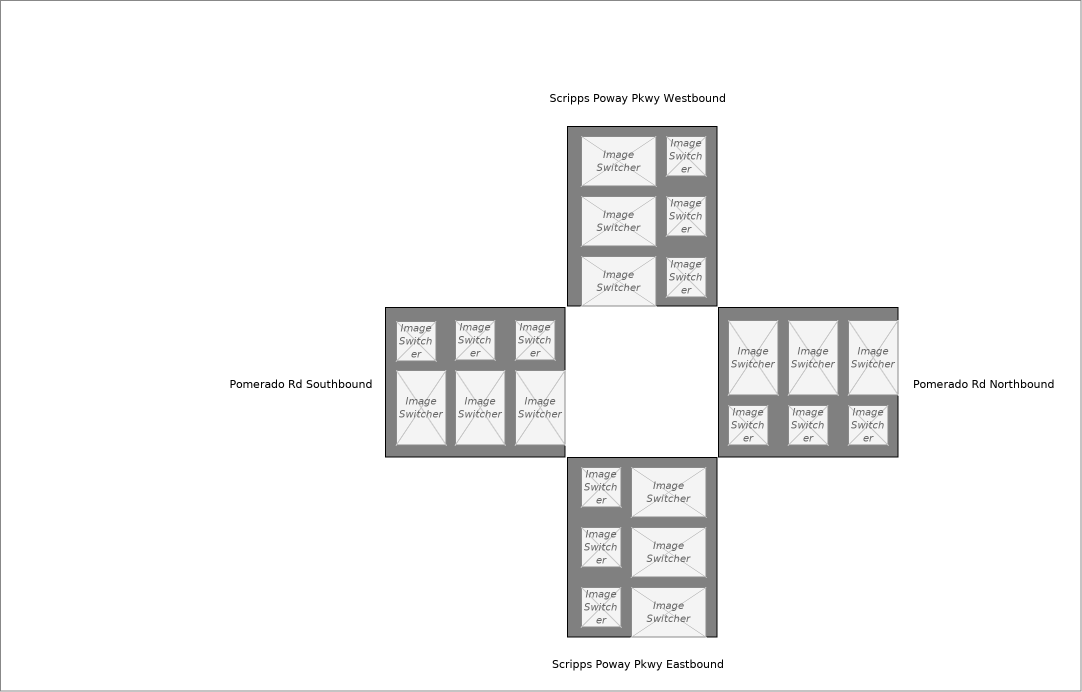
VISUALIZATION Initial_Intersection_Visualization  // 1082x692
    Group (203,71 879x566)
        Group (182,55 513x511)
            Group (182,331 150x180)
                RoundedRectangle (0,0 150x180)
                ImageSwitcher (64,70 75x50), variable: MAIN.fb_Major_Street_Forward_Phase_6.b_Yellow_Signal_Active, behaviour: TOGGLE
                ImageSwitcher (64,130 75x50), variable: MAIN.fb_Major_Street_Forward_Phase_6.b_Green_Signal_Active, behaviour: TOGGLE
                ImageSwitcher (64,10 75x50), variable: MAIN.fb_Major_Street_Forward_Phase_6.b_Red_Signal_Active, behaviour: TOGGLE
                ImageSwitcher (14,10 40x40), variable: MAIN.fb_Major_Street_Left_Turn_Phase_1.b_Red_Signal_Active, behaviour: TOGGLE
                ImageSwitcher (14,70 40x40), variable: MAIN.fb_Major_Street_Left_Turn_Phase_1.b_Yellow_Signal_Active, behaviour: TOGGLE
                ImageSwitcher (14,130 40x40), variable: MAIN.fb_Major_Street_Left_Turn_Phase_1.b_Green_Signal_Active, behaviour: TOGGLE
            Group (333,181 180x150)
                RoundedRectangle (0,0 180x150)
                Group (10,13 170x125)
                    ImageSwitcher (0,0 50x75), variable: MAIN.fb_Minor_Street_Forward_Phase_4.b_Red_Signal_Active, behaviour: TOGGLE
                    ImageSwitcher (60,0 50x75), variable: MAIN.fb_Minor_Street_Forward_Phase_4.b_Yellow_Signal_Active, behaviour: TOGGLE
                    ImageSwitcher (120,0 50x75), variable: MAIN.fb_Minor_Street_Forward_Phase_4.b_Green_Signal_Active, behaviour: TOGGLE
                    ImageSwitcher (0,85 40x40), variable: MAIN.fb_Minor_Street_Left_Turn_Phase_7.b_Red_Signal_Active, behaviour: TOGGLE
                    ImageSwitcher (60,85 40x40), variable: MAIN.fb_Minor_Street_Left_Turn_Phase_7.b_Yellow_Signal_Active, behaviour: TOGGLE
                    ImageSwitcher (120,85 40x40), variable: MAIN.fb_Minor_Street_Left_Turn_Phase_7.b_Green_Signal_Active, behaviour: TOGGLE
            RoundedRectangle (0,181 180x150)
            Group (11,194 169x125)
                ImageSwitcher (119,50 50x75), variable: MAIN.fb_Minor_Street_Forward_Phase_8.b_Red_Signal_Active, behaviour: TOGGLE
                ImageSwitcher (0,50 50x75), variable: MAIN.fb_Minor_Street_Forward_Phase_8.b_Green_Signal_Active, behaviour: TOGGLE
                ImageSwitcher (59,50 50x75), variable: MAIN.fb_Minor_Street_Forward_Phase_8.b_Yellow_Signal_Active, behaviour: TOGGLE
                ImageSwitcher (119,0 40x40), variable: MAIN.fb_Minor_Street_Left_Turn_Phase_3.b_Red_Signal_Active, behaviour: TOGGLE
                ImageSwitcher (59,0 40x40), variable: MAIN.fb_Minor_Street_Left_Turn_Phase_3.b_Yellow_Signal_Active, behaviour: TOGGLE
                ImageSwitcher (0,1 40x40), variable: MAIN.fb_Minor_Street_Left_Turn_Phase_3.b_Green_Signal_Active, behaviour: TOGGLE
            Group (182,0 150x180)
                RoundedRectangle (0,0 150x180)
                Group (14,10 125x170)
                    ImageSwitcher (0,120 75x50), variable: MAIN.fb_Major_Street_Forward_Phase_2.b_Red_Signal_Active, behaviour: TOGGLE
                    ImageSwitcher (0,60 75x50), variable: MAIN.fb_Major_Street_Forward_Phase_2.b_Yellow_Signal_Active, behaviour: TOGGLE
                    ImageSwitcher (0,0 75x50), variable: MAIN.fb_Major_Street_Forward_Phase_2.b_Green_Signal_Active, behaviour: TOGGLE
                    ImageSwitcher (85,121 40x40), variable: MAIN.fb_Major_Street_Left_Turn_Phase_5.b_Red_Signal_Active, behaviour: TOGGLE
                    ImageSwitcher (85,60 40x40), variable: MAIN.fb_Major_Street_Left_Turn_Phase_5.b_Yellow_Signal_Active, behaviour: TOGGLE
                    ImageSwitcher (85,0 40x40), variable: MAIN.fb_Major_Street_Left_Turn_Phase_5.b_Green_Signal_Active, behaviour: TOGGLE
        Label (337,0 196x55), "Scripps Poway Pkwy Westbound"
        Label (683,286 196x55), "Pomerado Rd Northbound"
        Label (0,286 196x55), "Pomerado Rd Southbound"
    Label (540,637 196x55), "Scripps Poway Pkwy Eastbound"
END_VISUALIZATION

(* stored: Version 1.1.0.1
   Visu Initial_Intersection_Visualization: Id {73742de4-a72e-44ef-b847-92b1b95797e4} *)
